{attribute 'linkalways'} 
{attribute 'no_explicit_call' := 'This FB is a CLASS and must be accessed using methods or properties'}
{attribute 'enable_dynamic_creation'}
FUNCTION_BLOCK Node_F_VN_InsertIntoContainer_TcVnVector4_USINT EXTENDS VisionNode
VAR
    aElement : _TcVnVector4_USINT;
    ipContainer : _ITcVnContainer;
    nIndex : _ULINT(0);
    hrPrev : _HRESULT(S_OK);
    hresult : _HRESULT(S_OK);
END_VAR

METHOD PUBLIC  Clone : I_Node
VAR
	pNode : POINTER TO Node_F_VN_InsertIntoContainer_TcVnVector4_USINT;
END_VAR
pNode := __NEW(Node_F_VN_InsertIntoContainer_TcVnVector4_USINT);
Clone := pNode^;
END_METHOD

METHOD FB_init : BOOL
VAR_INPUT
	bInitRetains : BOOL; // if TRUE, the retain variables are initialized (warm start / cold start)
	bInCopyCode : BOOL;  // if TRUE, the instance afterwards gets moved into the copy code (online change)
END_VAR
AddInput('aElement', aElement);
AddInput('ipContainer', ipContainer);
AddParameter('nIndex', nIndex);
AddInput('hrPrev', hrPrev);
AddOutput('ipContainer', ipContainer);
AddOutput('hresult',hresult);
END_METHOD

METHOD PROTECTED OnExecute
hresult.Value := F_VN_InsertIntoContainer_TcVnVector4_USINT(
    aElement := aElement.Value,
    ipContainer := ipContainer.Value,
    nIndex := nIndex.Value,
    hrPrev:= hrPrev.Value);
END_METHOD

METHOD PUBLIC PreExecutionCheck
VAR_INPUT
	Check : I_PreExecutionChecks;
END_VAR
Check.IsTrue(ipContainer.IsValid, 'ipContainer must be a valid container');
Check.IsTrue(ipContainer.IsType(TC_GLOBAL_CONST_LIST.ContainerType_Vector_TcVnVector4_USINT), 'ipContainer contains incorrect type');
END_METHOD

END_FUNCTION_BLOCK

(* stored: Version 1.1.0.1, ProductVersion 3.1.4026.13
   POU Node_F_VN_InsertIntoContainer_TcVnVector4_USINT: Id {b692f61a-eba5-4488-9d39-e73936fa847f}, SpecialFunc None
   Folder Constructor: Id {4efeb039-1856-41c5-88bc-3092a4d0391e}
   Method Clone: Id {102dc4f1-fc2d-4d68-b6a9-8aaab76ee724}
   Method FB_init: Id {12dce55d-bbf5-4b5b-8b9f-b0e5ca1d0168}
   Method OnExecute: Id {0c904a6d-ee19-4fc3-9db9-be805801df66}
   Method PreExecutionCheck: Id {18b59ee7-bc29-4ccf-9250-9198c0cca0d2} *)
